// TwinCAT 3 PLC project simple
// ProgramVersion: 3.1.4023.0
// libraries:
//   Tc2_MC2, * (Beckhoff Automation GmbH)
//   Tc2_MC2_Drive, * (Beckhoff Automation GmbH)
//   Tc2_NC, * (Beckhoff Automation GmbH)
//   Tc2_Standard, * (Beckhoff Automation GmbH)
//   Tc2_System, * (Beckhoff Automation GmbH)
//   Tc3_Module, * (Beckhoff Automation GmbH)
//   VisuSymbols,3.5.10.0,System
// project tree:
//   / GlobalTextList.TcGTLO, PlcTask.TcTTO, Visualization Manager.TcVMO (not stored)
//   GVLs/ Controls_GVL.TcGVL, GVL_axisContr.TcGVL, GVL_NC.TcGVL, GVL_Sensors.TcGVL
//   POUs/ MAIN.TcPOU, POU_MainFunc.TcPOU, POU_NCPowerOn.TcPOU, POU_XaxisCtrl.TcPOU
//   VISUs/ Visualization.TcVIS
// real-time tasks:
//   TASK PlcTask: cycle T#10ms, priority 20, ADS port 350
// motion (NC):
//   TASK NC-Task 1 SAF: cycle T#2ms, priority 4, ADS port 501
//   TASK NC-Task 1 SVB: cycle T#10ms, priority 8, ADS port 511
//   AXIS Axis X (id 1)
//     Dynamic: Acceleration=252.5, Deceleration=252.5, Jerk=31878
//     Velo: Maximum=200
//     PositionAreaControl: Enable=false
//     OtherSettings: AllowMotionCmdToSlave=true
//     encoder EncType=4
//       EncPara: MaxCount=#x0000ffff
//         Inc: RefSoftSyncMask=#x0000ffff
//     drive DrvType=24
//       Analog: VeloReferenz=200, TorqueSetpointScale=10, ScaleFactorActTorque=0.1
//       TimeComp: TaskDelayCycles=1
//     controller CtrType=1
//       CtrPara: PriorControlFactor=1
//         PosDiffControl: Enable=false, Range=8, Time=0.08
//         Observer: BandWidth=20
// I/O:
//   DEVICE Device 3 (EtherCAT), AmsNetId 5.58.164.20.4.1
//     Term 1 (EK1914) [EK1914, 2 Ch. Safety Input/Output 24V,  TwinSAFE]
//       modules: Module 1 (FSOE), Module 2 (DIO)
//       Term 2 (EL1809) [EL1809 16Ch. Dig. Input 24V, 3ms]
//       Term 3 (EL7031) [EL7031 1Ch. Stepper motor output stage (24V, 1.5A)]
//       Term 4 (EL2008) [EL2008 8Ch. Dig. Output 24V, 0.5A]
//       Term 5 (EL1008) [EL1008 8Ch. Dig. Input 24V, 3ms]
//       Term 15 (EL9011) [EL9011 End Terminal]
// variable links:
//   NC-Task 1 SAF/Axes/Axis X <-> Device 3 (EtherCAT)/Term 1 (EK1914)/Term 3 (EL7031)
//     Drive/Inputs/In/nState1 @bit 3 <-> STM Status/Status/Error
//     Drive/Inputs/In/nState1 @bit 5 <-> STM Status/Status/Moving negative
//     Drive/Inputs/In/nState1 @bit 4 <-> STM Status/Status/Moving positive
//     Drive/Inputs/In/nState1 @bit 1 <-> STM Status/Status/Ready
//     Drive/Inputs/In/nState1 <-> STM Status/Status/Ready to enable
//     Drive/Inputs/In/nState1 @bit 6 <-> STM Status/Status/Torque reduced
//     Drive/Inputs/In/nState1 @bit 2 <-> STM Status/Status/Warning
//     Drive/Inputs/In/nState2 @bit 3 <-> STM Status/Status/Digital input 1
//     Drive/Inputs/In/nState2 @bit 4 <-> STM Status/Status/Digital input 2
//     Drive/Inputs/In/nState2 @bit 5 <-> STM Status/Status/Sync error
//     Drive/Inputs/In/nState2 @bit 7 <-> STM Status/Status/TxPDO Toggle
//     Drive/Inputs/In/nState4 @bit 1 <-> WcState/InputToggle
//     Drive/Inputs/In/nState4 <-> WcState/WcState
//     Drive/Outputs/Out/nCtrl1 <-> STM Control/Control/Enable
//     Drive/Outputs/Out/nCtrl1 @bit 2 <-> STM Control/Control/Reduce torque
//     Drive/Outputs/Out/nCtrl1 @bit 1 <-> STM Control/Control/Reset
//     Drive/Outputs/Out/nDataOut2[0] <-> STM Velocity/Velocity
//     Enc/Inputs/In/nDataIn1[0] <-> ENC Status compact/Counter value
//     Enc/Inputs/In/nDataIn2[0] <-> ENC Status compact/Latch value
//     Enc/Inputs/In/nState1 @bit 4 <-> ENC Status compact/Status/Counter overflow
//     Enc/Inputs/In/nState1 @bit 3 <-> ENC Status compact/Status/Counter underflow
//     Enc/Inputs/In/nState1 @bit 1 <-> ENC Status compact/Status/Latch extern valid
//     Enc/Inputs/In/nState1 @bit 2 <-> ENC Status compact/Status/Set counter done
//     Enc/Inputs/In/nState2 @bit 4 <-> ENC Status compact/Status/Status of extern latch
//     Enc/Inputs/In/nState2 @bit 5 <-> ENC Status compact/Status/Sync error
//     Enc/Inputs/In/nState2 @bit 7 <-> ENC Status compact/Status/TxPDO Toggle
//     Enc/Inputs/In/nState4 @bit 1 <-> WcState/InputToggle
//     Enc/Inputs/In/nState4 <-> WcState/WcState
//     Enc/Outputs/Out/nCtrl1 @bit 3 <-> ENC Control compact/Control/Enable latch extern on negative edge
//     Enc/Outputs/Out/nCtrl1 @bit 1 <-> ENC Control compact/Control/Enable latch extern on positive edge
//     Enc/Outputs/Out/nCtrl1 @bit 2 <-> ENC Control compact/Control/Set counter
//     Enc/Outputs/Out/nDataOut1[0] <-> ENC Control compact/Set counter value
//   simple/simple Instance <-> Device 3 (EtherCAT)/Term 1 (EK1914)/Term 2 (EL1809)
//     PlcTask Inputs/Controls_GVL.BendDown <-> Channel 7/Input
//     PlcTask Inputs/Controls_GVL.CloseGripp <-> Channel 9/Input
//     PlcTask Inputs/Controls_GVL.Estop <-> Channel 3/Input
//     PlcTask Inputs/Controls_GVL.ManualIn <-> Channel 4/Input
//     PlcTask Inputs/Controls_GVL.RLInp <-> Channel 6/Input
//     PlcTask Inputs/Controls_GVL.RRInp <-> Channel 2/Input
//     PlcTask Inputs/Controls_GVL.Reset <-> Channel 5/Input
//     PlcTask Inputs/Controls_GVL.StandUp <-> Channel 8/Input
//   simple/simple Instance <-> Device 3 (EtherCAT)/Term 1 (EK1914)/Term 4 (EL2008)
//     PlcTask Outputs/Controls_GVL.BDout <-> Channel 4/Output
//     PlcTask Outputs/Controls_GVL.CGout <-> Channel 6/Output
//     PlcTask Outputs/Controls_GVL.Light <-> Channel 7/Output
//     PlcTask Outputs/Controls_GVL.ManualMo <-> Channel 1/Output
//     PlcTask Outputs/Controls_GVL.RotateLeft <-> Channel 3/Output
//     PlcTask Outputs/Controls_GVL.RotateRight <-> Channel 2/Output
//     PlcTask Outputs/Controls_GVL.SUout <-> Channel 5/Output
//   simple/simple Instance <-> NC-Task 1 SAF/Axes/Axis X
//     PlcTask Inputs/GVL_NC.AxisX.NcToPlc <-> Outputs/ToPlc
//     PlcTask Outputs/GVL_NC.AxisX.PlcToNc <-> Inputs/FromPlc

CONFIGURATION simple
    RESOURCE PLC ON TwinCAT3
        TASK PlcTask(INTERVAL := T#10ms, PRIORITY := 20);
        PROGRAM MAIN WITH PlcTask : MAIN;
    END_RESOURCE
END_CONFIGURATION

// ---- GVLs/Controls_GVL.TcGVL
VAR_GLOBAL
	Light			AT %Q*	:BOOL;		//Digital Input on Ek1914 card 1. 'AT %I' shows it is an hardware input, ':BOOL;' declares the type, in this case, it's a Boolean. 
	ManualMo        AT %Q*  :BOOL;
	RotateRight 	AT %Q*  :BOOL;
	RRInp 			AT %I*  :BOOL;
	RotateLeft 		AT %Q*  :BOOL;
	RLInp			AT %I*  :BOOL;
	Reset           AT %I* 	:BOOL;
	Estop  			AT %I* 	:BOOL;
	ManualIn 		AT %I*  :BOOL;
	BendDown		AT %I*  :BOOL;
	StandUp			AT %I*  :BOOL;
	CloseGripp		AT %I*  :BOOL;
	BDout			AT %Q*  :BOOL;
	SUout			AT %Q*  :BOOL;
	CGout			AT %Q*  :BOOL;
	EstopOut		AT %Q*  :BOOL;
	IRSensor		AT %I*  :BOOL;
	plctonc			AT %Q*  :PLCTONC_AXLESTRUCT_CTRL;
	nctoplc 		AT %I*  :NCTOPLC_AXLESTRUCT_STATE;
	Position: INT;
END_VAR

// ---- GVLs/GVL_axisContr.TcGVL
VAR_GLOBAL
	XAxisEnable:BOOL;
	XAxisJogPos:BOOL;
	XAxisJogNeg:BOOL;
	
END_VAR

// ---- GVLs/GVL_NC.TcGVL
VAR_GLOBAL
	AxisX:AXIS_REF;
	AxisXStatus:ST_AxisStatus;
	
END_VAR

// ---- GVLs/GVL_Sensors.TcGVL
VAR_GLOBAL
	XAxisLimitSwPos AT %I* :BOOL;
	XAxisLimitSwNeg AT %I* :BOOL;
END_VAR

// ---- POUs/MAIN.TcPOU
PROGRAM MAIN
VAR
	Ladder : POU_MainFunc;
	Motor: POU_NCPowerOn;
	ReadXAxisStatus:MC_ReadStatus;
	poweraxis: MC_PowerStepper;
	resetaxis: MC_Reset;
	stopaxis: MC_Stop;
	MoveVelocity: MC_MoveVelocity;
	direction: MC_Direction;
	SetVel: MC_MoveAbsolute;
	
	
END_VAR


	
	
Ladder();
motor();

END_PROGRAM

// ---- POUs/POU_MainFunc.TcPOU
FUNCTION_BLOCK POU_MainFunc
VAR_INPUT
END_VAR
VAR_OUTPUT
END_VAR
VAR
	go: BOOL; //local variable to start the program and modes
	TON_0: TON;
	timepass: TIME;
	TimerAmount: TIME:= T#340MS; //this is a specific value type, time of 340ms
	timer2: BOOL;
	Timer1: BOOL;
	TON_1: TON;
	InManual: BOOL;
	Motor: MC_Power;
	onMotor: BOOL;
	Motormove: MC_MoveVelocity;
END_VAR

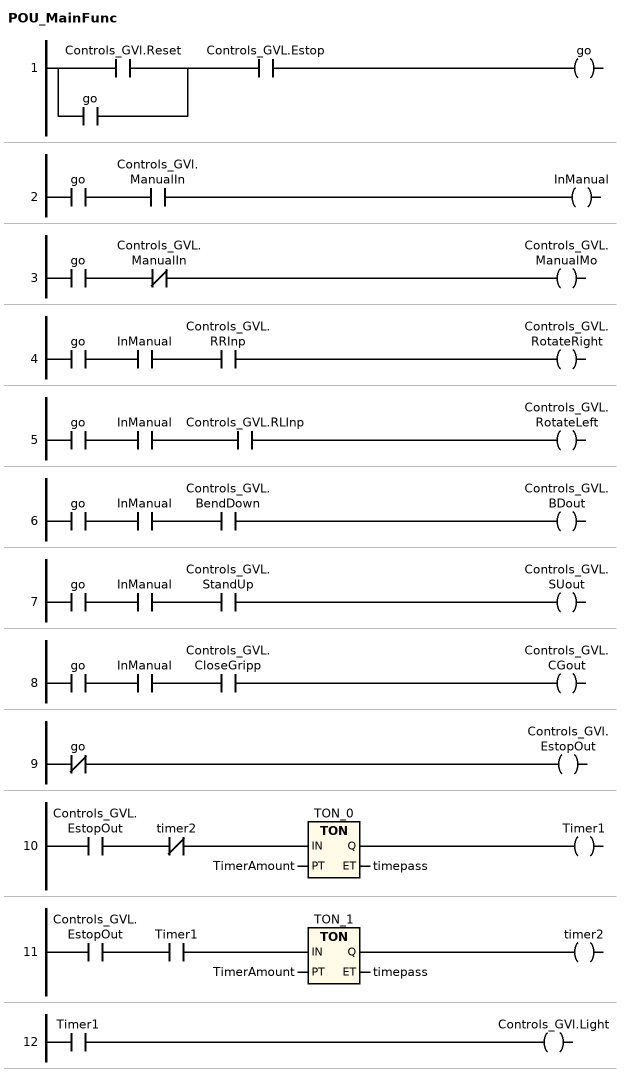
// NETWORK 1
go := (Controls_GVl.Reset OR go) AND Controls_GVL.Estop;

// NETWORK 2
InManual := go AND Controls_GVl.ManualIn;

// NETWORK 3
Controls_GVL.ManualMo := go AND NOT Controls_GVL.ManualIn;

// NETWORK 4
Controls_GVL.RotateRight := go AND InManual AND Controls_GVL.RRInp;

// NETWORK 5
Controls_GVL.RotateLeft := go AND InManual AND Controls_GVL.RLInp;

// NETWORK 6
Controls_GVL.BDout := go AND InManual AND Controls_GVL.BendDown;

// NETWORK 7
Controls_GVL.SUout := go AND InManual AND Controls_GVL.StandUp;

// NETWORK 8
Controls_GVL.CGout := go AND InManual AND Controls_GVL.CloseGripp;

// NETWORK 9
Controls_GVl.EstopOut := NOT go;

// NETWORK 10
TON_0(IN := Controls_GVL.EstopOut AND NOT timer2, PT := TimerAmount, ET => timepass); // TON
Timer1 := TON_0.Q;

// NETWORK 11
TON_1(IN := Controls_GVL.EstopOut AND Timer1, PT := TimerAmount, ET => timepass); // TON
timer2 := TON_1.Q;

// NETWORK 12
Controls_GVl.Light := Timer1;

END_FUNCTION_BLOCK

// ---- POUs/POU_NCPowerOn.TcPOU
FUNCTION_BLOCK POU_NCPowerOn
VAR_INPUT
END_VAR
VAR_OUTPUT
END_VAR
VAR
	XAxisPowerOn: MC_Power;
	GoMotor: MC_MoveVelocity;
	direction: MC_Direction;
	TRUEB: BOOL;
	MoveDistance: MC_MoveModulo;
	MoveBack: MC_MoveModulo;
	DoneT: BOOL;
END_VAR

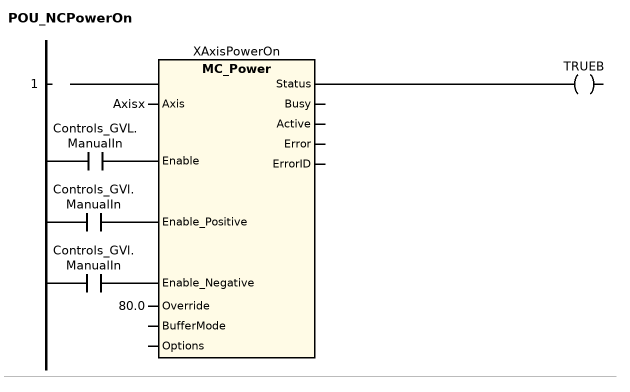
// NETWORK 1
XAxisPowerOn(
    Axis := Axisx,
    Enable := Controls_GVL.ManualIn,
    Enable_Positive := Controls_GVl.ManualIn,
    Enable_Negative := Controls_GVl.ManualIn,
    Override := 80.0); // MC_Power
TRUEB := XAxisPowerOn.Status;

END_FUNCTION_BLOCK

// ---- POUs/POU_XaxisCtrl.TcPOU
FUNCTION_BLOCK POU_XaxisCtrl
VAR_INPUT
END_VAR
VAR_OUTPUT
END_VAR
VAR
END_VAR

// NETWORK 1

END_FUNCTION_BLOCK

// ---- VISUs/Visualization.TcVIS
VISUALIZATION Visualization  // 2x2
END_VISUALIZATION
